// TIA Portal V20 export
TYPE "typeCmHmiInterfaceSoftCam"
// stored: Access Published, Namespace Unit1.Em8
   STRUCT
      thicknessAxisZ : "Unit1.Em8.typeCmHmiInterfaceSoftCamthicknessAxisZ";
   END_STRUCT;
END_TYPE
